FUNCTION_BLOCK FB_EX_Example
//////////////////
// 
//////////////////
VAR CONSTANT PERSISTENT
	// Characteristics of the object (Same for all instances)
	
END_VAR

VAR_INPUT PERSISTENT
	// Parameters of the Object (instance specific) 
	
END_VAR

VAR_OUTPUT
	//Child objects
	
END_VAR
VAR
	//M_METHOD2 VARIABLES//
	
	
	//M_METHOD2 VARIABLES//
	
	
	//M_METHOD3 VARIABLES//
	
	
	//GET/SET PROPERTY MANAGEMENT//
	
	
END_VAR

END_FUNCTION_BLOCK

(* stored: Version 1.1.0.1, ProductVersion 3.1.4024.6
   POU FB_EX_Example: Id {9b0238b6-50ca-4292-af2d-6bdc793c8987}, SpecialFunc None *)
